# B&R Automation Studio project MySQLConnectorDemo
Automation Studio 4.12.6.106

## Configuration Config1

CPU X20CP3586, AutomationRuntime I4.93, Build 6.3.0, Vc 

### Task classes (Cpu.sw)
```
Cyclic#4:
  CmdGenerat <- MySQLInserter.CmdGenerator.prg
  Demo <- MySQLInserter.Demo.prg
  SqlWriter <- MySQLInserter.SqlWriter.prg
Binaries: udbdef, FWRules, TCData, sysconf, Role, User, iomap, ashwd, asfw, arconfig, ashwac
Libraries: AsBrStr, sys_lib, runtime, LxVar, asstring, astime, asieccon, BrRand, brsystem, standard
```

### Hardware
```
X20CP3586 : X20CP3586 v1.10.0.0
  Connector IF2:
    ActivateDevice = 1
    Mode = Manual
    InternetAddress = 192.168.0.200
    SubnetMask = 255.255.255.0
    ActivateSnmp = 2
  ConfigurationID = MySQLConnectorDemo_Config1
  RemanentGlobalPvSize = 80960
  FileDevice1
  FileDeviceName1 = USER
  FileDevicePath1 = USER_PATH
  ActivateOpcUa = 1
  OpcUaInformationModels_PV_Version = 1
```

### Config.mpdatabasecore - X20CP3586/mappServices/Config.mpdatabasecore
```
Element gDatabaseCore (Type=mpdatabasecore)
  mapp.Database.Core:
    Name = wn_9
    UserName = newuser
    Password = 123456
    PortNumber = 85
    DBQueries:
      [0]:
        Name = RdByTime
        Type = Custom
          Query = {&pv[gSqlStr]}
          Columns = SingleColumns
            [0]:
              Column = rdFloat1
              PV = ::SqlReader:RdBuffer.rdFloat1[]
            [1]:
              Column = rdFloat2
              PV = ::SqlReader:RdBuffer.rdFloat2[]
            [2]:
              Column = rdFloat3
              PV = ::SqlReader:RdBuffer.rdFloat3[]
      [1]:
        Name = RdByName
        Type = Custom
          Query = {&pv[gSqlStr]}
          Columns:
            PV = 
```

## Logical view

Binary libraries used (declarations not repeated): operator, runtime, astime, AsIecCon, AsBrStr, sys_lib, asstring, brsystem, standard, MpDatabase 5.24.3, BrRand

### Package Logical/Libraries - Global libraries

### GlobalMySQL.var
```iecst
VAR
	gMySQLInserter : MySQLInserter_typ;
END_VAR
VAR CONSTANT
	TASK_SIZE : USINT := 4;
	TASK_SIZE_MINUS_ONE : USINT := TASK_SIZE-1;
	INTERFACE_SIZE : USINT := 1;
	INTERFACE_SIZE_MINUS_ONE : USINT := INTERFACE_SIZE-1;
	CMD_STR_SIZE : UINT := 4000;
	SQL_NAME_STR_SIZE : USINT := 10;
	DATA_SIZE : USINT := 100;
	DATA_SIZE_MINUS_ONE : USINT := DATA_SIZE-1;
END_VAR
```

### GlobalMySQL.typ
```iecst
TYPE
	MySQLInserter_typ : 	STRUCT
		Command : MySQLInserterCommand_typ;
		Input : MySQLInserterInput_typ;
		Status : MySQLInserterStatus_typ;
		Config : MySQLInserterConfig_typ;
		ExternalCom : MySQLInserterExternalCom_typ;
		_Internal : MySQLInserterInternal_typ;
	END_STRUCT;
	MySQLInserterCommand_typ : 	STRUCT
		Enable : BOOL;
		Reset : BOOL;
	END_STRUCT;
	MySQLInserterInput_typ : 	STRUCT
		TaskTrig : ARRAY[0..TASK_SIZE_MINUS_ONE]OF BOOL;
	END_STRUCT;
	MySQLInserterStatus_typ : 	STRUCT
		BufferNum : ARRAY[0..INTERFACE_SIZE_MINUS_ONE]OF USINT;
		Connected : BOOL;
		Task : ARRAY[0..TASK_SIZE_MINUS_ONE]OF TaskStatus_typ;
	END_STRUCT;
	MySQLInserterConfig_typ : 	STRUCT
		TaskSetting : ARRAY[0..TASK_SIZE_MINUS_ONE]OF TaskSetting_typ;
		LostTimeMs : UDINT; (*Connect lost time*)
	END_STRUCT;
	MySQLInserterInternal_typ : 	STRUCT
		TaskCmdStr : ARRAY[0..TASK_SIZE_MINUS_ONE]OF STRING[CMD_STR_SIZE];
	END_STRUCT;
	MySQLInserterExternalCom_typ : 	STRUCT
		StrCmd : ARRAY[0..INTERFACE_SIZE_MINUS_ONE]OF STRING[CMD_STR_SIZE];
		Counter : ARRAY[0..INTERFACE_SIZE_MINUS_ONE]OF UDINT;
		HeartBeat : ARRAY[0..INTERFACE_SIZE_MINUS_ONE]OF UDINT;
	END_STRUCT;
	DataSetting_typ : 	STRUCT
		Name : STRING[SQL_NAME_STR_SIZE];
		Type : STRING[SQL_NAME_STR_SIZE];
		DataAddr : UDINT;
		DataSize : USINT; (*VARCHAR需要设置，DATETIME推荐设置*)
		Digital : USINT; (*仅FLOAT有效：
保留小数点位数*)
		ManualTime : BOOL; (*仅DATETIME有效:
0：自动生成TimeStamp
1：外部给出TimeStamp*)
		MissingCheck : BOOL; (*仅INT有效:(关联数据，外部请勿操作)
0：关闭
1：开启，默认自增1，用于检查是否漏写*)
		AutoIncrement : BOOL; (*mysql属性AUTO_INCREMENT*)
		NotNull : BOOL; (*mysql属性NOT NULL*)
		PrimaryKey : BOOL; (*mysql属性PRIMARY KEY*)
	END_STRUCT;
	MySQLInserterTask_typ : 	STRUCT
		Setting : TaskSetting_typ;
		Status : TaskStatus_typ;
	END_STRUCT;
	TaskStatus_typ : 	STRUCT
		Err : USINT;
		ErrMsg : STRING[64];
		CacheCount : USINT;
	END_STRUCT;
	TaskSetting_typ : 	STRUCT
		TrigMode : USINT; (*0：外部上升沿触发
1：按照采样时间自动触发*)
		IntervalTimeMs : UINT; (*采样间隔时间ms，最好不要<1000，最好是1000的整数倍*)
		DbName : STRING[SQL_NAME_STR_SIZE];
		TableName : STRING[SQL_NAME_STR_SIZE];
		CacheSize : USINT; (*缓存大小，设置合并插入*)
		WritePrimaryKey : USINT; (*是否写入主键*)
		DataSetting : ARRAY[0..DATA_SIZE_MINUS_ONE]OF DataSetting_typ;
	END_STRUCT;
END_TYPE
```

### Program Logical/MySQLInserter/CmdGenerator (ANSIC)

#### Variables.var - Local variables
```iecst
VAR
	InsCfg : REFERENCE TO MySQLInserterConfig_typ;
	InsSts : REFERENCE TO MySQLInserterStatus_typ;
	InsInter : REFERENCE TO MySQLInserterInternal_typ;
	InsInput : REFERENCE TO MySQLInserterInput_typ;
	InsCmd : REFERENCE TO MySQLInserterCommand_typ;
	u8idx : USINT;
	strBuffer : ARRAY[0..TASK_SIZE_MINUS_ONE] OF STRING[CMD_STR_SIZE];
	RTInfo_0 : RTInfo;
	accTimeUs : ARRAY[0..TASK_SIZE_MINUS_ONE] OF UDINT;
	firstScan : BOOL;
END_VAR
```

#### Main.c - Init, cyclic, exit code
```c
#include <bur/plctypes.h>
#include "SqlMaker.h"
#ifdef _DEFAULT_INCLUDES
	#include <AsDefault.h>
#endif

void _INIT ProgramInit(void)
{
	// Insert code here
	InsCfg = &gMySQLInserter.Config;
	InsSts = &gMySQLInserter.Status;
	InsInter = &gMySQLInserter._Internal;
	InsInput = &gMySQLInserter.Input;
	InsCmd = &gMySQLInserter.Command;
	firstScan = 1;
}

void _CYCLIC ProgramCyclic(void)
{
	// Insert code here
	if (0 == InsCmd->Enable) {
		return;
	}

	if (InsCmd->Reset) {
		firstScan = 1;
	}

	/* 获取线程信息 */
	RTInfo_0.enable = 1;
	RTInfo(&RTInfo_0);

	if (firstScan) {
		for (u8idx = 0; u8idx < TASK_SIZE ; u8idx++) {
			MakeCreateTableSql(strBuffer[u8idx], CMD_STR_SIZE, &InsCfg->TaskSetting[u8idx]);
			brsmemcpy((UDINT)InsInter->TaskCmdStr[u8idx], (UDINT)strBuffer[u8idx], CMD_STR_SIZE);
			InsSts->Task[u8idx].CacheCount = 0; // Cache清0
		}
		firstScan = 0;
		return;
	}

	for (u8idx = 0; u8idx < TASK_SIZE ; u8idx++) {
		// 定时触发模式
		if (1 == InsCfg->TaskSetting[u8idx].TrigMode) {
			if (InsCfg->TaskSetting[u8idx].IntervalTimeMs * 1000 > RTInfo_0.cycle_time && RTInfo_0.cycle_time != 0) {
				accTimeUs[u8idx] = accTimeUs[u8idx] + RTInfo_0.cycle_time;
				if (accTimeUs[u8idx] >= InsCfg->TaskSetting[u8idx].IntervalTimeMs * 1000){
					// 计时到，采集一次数据
					MakeInsertSql(strBuffer[u8idx], CMD_STR_SIZE, &InsCfg->TaskSetting[u8idx], &InsSts->Task[u8idx]);
					accTimeUs[u8idx] = 0;
				}
			} else {
				InsSts->Task[u8idx].Err = 1;
				strcpy(InsSts->Task[u8idx].ErrMsg, "Sampling interval is less than task cycle time.");
			}
		// 手动触发模式
		}else if (0 == InsCfg->TaskSetting[u8idx].TrigMode) {
			if (1 == InsInput->TaskTrig[u8idx]) {
				InsInput->TaskTrig[u8idx] = 0;
				MakeInsertSql(strBuffer[u8idx], CMD_STR_SIZE, &InsCfg->TaskSetting[u8idx], &InsSts->Task[u8idx]);
			}
		}
		// 到达cache_size大小，自动封包
		if (0 == InsSts->Task[u8idx].CacheCount) {
			// memset((UDINT)InsInter->TaskCmdStr[u8idx], 0, CMD_STR_SIZE);
			brsmemcpy((UDINT)InsInter->TaskCmdStr[u8idx], (UDINT)strBuffer[u8idx], CMD_STR_SIZE);
		}
	}
}

void _EXIT ProgramExit(void)
{
	// Insert code here

}
```

#### SqlMaker.h
```c
#ifndef SQLMAKER_H
#define SQLMAKER_H

#include <bur/plctypes.h>
#include <string.h>
#include <LxVar.h>

#ifdef _DEFAULT_INCLUDES
	#include <AsDefault.h>
#endif

void MakeInsertSql(STRING* sqlBuffer, UDINT bufferSize, TaskSetting_typ* taskSetting, TaskStatus_typ* taskStatus);
void MakeCreateTableSql(STRING* sqlBuffer, UDINT bufferSize, TaskSetting_typ* taskSetting);
UDINT CreateMySQLDateTimeStamp(STRING *pOutputString);

#endif // SQLMAKER_H
```

#### SqlMaker.c
```c
#include "SqlMaker.h"

void MakeInsertSql(STRING* sqlBuffer, UDINT bufferSize, TaskSetting_typ* taskSetting, TaskStatus_typ* taskStatus)
{
	// Calc data size
	if (0 == sizeof(taskSetting->DataSetting[0])) {
		return;
	}
	int dataSize = sizeof(taskSetting->DataSetting)/sizeof(taskSetting->DataSetting[0]);

	if (dataSize < 1) {
		return;
	}

	// Start building the SQL command
	if (0 == taskStatus->CacheCount) {
		memset((char*)sqlBuffer, 0, bufferSize);
		strcat((char*)sqlBuffer, "INSERT INTO ");
		strcat((char*)sqlBuffer, taskSetting->DbName);
		strcat((char*)sqlBuffer, ".");
		strcat((char*)sqlBuffer, taskSetting->TableName);
		strcat((char*)sqlBuffer, " (");

		// Add column names
		for (int i = 0; i < dataSize; ++i) {
			if (taskSetting->DataSetting[i].Name[0] == '\0') break;
			if (taskSetting->WritePrimaryKey == 0 && taskSetting->DataSetting[i].PrimaryKey == 1) {
				continue;
			}
			strcat((char*)sqlBuffer, taskSetting->DataSetting[i].Name);
			if (i < (dataSize - 1) && taskSetting->DataSetting[i+1].Name[0] != '\0') {
				strcat((char*)sqlBuffer, ",");
			}
		}
		strcat((char*)sqlBuffer, ") VALUES");
	}

	strcat((char*)sqlBuffer, "(");
	STRING tempStr[32];
	FB_Real2Str_typ FB_Real2Str_0;
	// Add value placeholders
	for (int i = 0; i < dataSize; ++i) {
		if (taskSetting->DataSetting[i].Name[0] == '\0') break;
		if (taskSetting->WritePrimaryKey == 0 && taskSetting->DataSetting[i].PrimaryKey == 1) {
			continue;
		}
		memset((char*)tempStr, 0, sizeof(tempStr));
		// Use '%s' for string, '%d' for int, etc. Here, just use '?' as placeholder
		if (strcmp(taskSetting->DataSetting[i].Type, "FLOAT") == 0) {
			// Type is FLOAT
			if (taskSetting->DataSetting[i].Digital != 0) {
				FB_Real2Str_0.digital = taskSetting->DataSetting[i].Digital;
				FB_Real2Str_0.rNum = *(REAL*)(taskSetting->DataSetting[i].DataAddr);
				FB_Real2Str(&FB_Real2Str_0);
				strcat((char*)tempStr, FB_Real2Str_0.strOut);
			}else {
				ftoa(*(REAL*)taskSetting->DataSetting[i].DataAddr, (UDINT)tempStr);
			}
			strcat((char*)sqlBuffer, (char*)tempStr);
		}
		else if (strcmp(taskSetting->DataSetting[i].Type, "INT") == 0) {
			// Type is INT
			if (1 == taskSetting->DataSetting[i].MissingCheck) {
				*(DINT*)taskSetting->DataSetting[i].DataAddr += 1;
			}
			itoa(*(DINT*)taskSetting->DataSetting[i].DataAddr, (UDINT)tempStr);
			strcat((char*)sqlBuffer, (char*)tempStr);
		}
		else if (strcmp(taskSetting->DataSetting[i].Type, "VARCHAR") == 0) {
			// Type is VARCHAR
			strcat((char*)sqlBuffer, (char*)taskSetting->DataSetting[i].DataAddr);
		}
		else if (strcmp(taskSetting->DataSetting[i].Type, "DATETIME") == 0) {
			// Type is DATETIME
			if (0 == taskSetting->DataSetting[i].ManualTime) {
				CreateMySQLDateTimeStamp(&tempStr);
				strcat((char*)sqlBuffer, (char*)tempStr);
			}else {
				strcat((char*)sqlBuffer, (char*)taskSetting->DataSetting[i].DataAddr);
			}
		}
		else {
			// Default case, treat as string
		}

		if (i < (dataSize - 1) && taskSetting->DataSetting[i+1].Name[0] != '\0') {
			strcat((char*)sqlBuffer, ",");
		}
	}
	strcat((char*)sqlBuffer, ")");
	if (taskStatus->CacheCount < (taskSetting->CacheSize - 1) && taskSetting->CacheSize != 0) {
		taskStatus->CacheCount = taskStatus->CacheCount + 1;
		strcat((char*)sqlBuffer, ",");
	} else {
		taskStatus->CacheCount = 0;
		strcat((char*)sqlBuffer, ";");
	}
}

void MakeCreateTableSql(STRING* sqlBuffer, UDINT bufferSize, TaskSetting_typ* taskSetting)
{
	if (0 == sizeof(taskSetting->DataSetting[0])) {
		return;
	}
	int dataSize = sizeof(taskSetting->DataSetting)/sizeof(taskSetting->DataSetting[0]);
	if (dataSize < 1) {
		return;
	}

	memset((char*)sqlBuffer, 0, bufferSize);
	strcat((char*)sqlBuffer, "CREATE TABLE IF NOT EXISTS ");
	strcat((char*)sqlBuffer, taskSetting->DbName);
	strcat((char*)sqlBuffer, ".");
	strcat((char*)sqlBuffer, taskSetting->TableName);
	strcat((char*)sqlBuffer, " (");

	for (int i = 0; i < dataSize; ++i) {
		if (taskSetting->DataSetting[i].Name[0] == '\0') {
			if (0 == i) {
				memset((char*)sqlBuffer, 0, bufferSize);
				return;
			}
			break;
		}
		strcat((char*)sqlBuffer, taskSetting->DataSetting[i].Name);
		strcat((char*)sqlBuffer, " ");
		strcat((char*)sqlBuffer, taskSetting->DataSetting[i].Type);

		// VARCHAR length
		if (strcmp(taskSetting->DataSetting[i].Type, "VARCHAR") == 0 && taskSetting->DataSetting[i].DataSize > 0) {
			char lenStr[8] = {0};
			strcat((char*)sqlBuffer, "(");
			itoa(taskSetting->DataSetting[i].DataSize, (UDINT)lenStr);
			strcat((char*)sqlBuffer, lenStr);
			strcat((char*)sqlBuffer, ")");
		}

		// Auto increment
		if (taskSetting->DataSetting[i].AutoIncrement) {
			strcat((char*)sqlBuffer, " AUTO_INCREMENT");
		}

		// NOT NULL
		if (taskSetting->DataSetting[i].NotNull) {
			strcat((char*)sqlBuffer, " NOT NULL");
		}

		// PRIMARY KEY
		if (taskSetting->DataSetting[i].PrimaryKey) {
			strcat((char*)sqlBuffer, " PRIMARY KEY");
		}

		if (i < (dataSize - 1) && taskSetting->DataSetting[i+1].Name[0] != '\0') {
			strcat((char*)sqlBuffer, ",");
		}
	}
	strcat((char*)sqlBuffer, ");");
}

UDINT CreateMySQLDateTimeStamp(STRING *pOutputString)
{
	STRING tempString[10];
	RTCtime_typ	RTC;

	/* Clear output string */
	memset(pOutputString, 0, sizeof(*pOutputString));
	/* Clear temp string */
	memset(&tempString, 0, sizeof(tempString));

	/* Get time */
	RTC_gettime(&RTC);

	/* copy in single quote */
	strcpy(pOutputString, "'");
	/* copy in year */
	itoa(RTC.year, (UDINT)tempString);
	strcat(pOutputString, tempString);
	/* add dash */
	strcat(pOutputString, "-");
	/* copy in month */
	itoa(RTC.month, (UDINT)tempString);
	strcat(pOutputString, tempString);
	/* add dash */
	strcat(pOutputString, "-");
	/* copy in day */
	itoa(RTC.day, (UDINT)tempString);
	strcat(pOutputString, tempString);

	/* add space */
	strcat(pOutputString, " ");

	/* copy in hour */
	itoa(RTC.hour, (UDINT)tempString);
	strcat(pOutputString, tempString);
	/* add colon */
	strcat(pOutputString, ":");
	/* copy in minutes */
	itoa(RTC.minute, (UDINT)tempString);
	strcat(pOutputString, tempString);
	/* add colon */
	strcat(pOutputString, ":");
	/* copy in seconds */
	itoa(RTC.second, (UDINT)tempString);
	strcat(pOutputString, tempString);
	/* copy in single quote */
	strcat(pOutputString, "'");

	return((UDINT)pOutputString);
}
```

### Program Logical/MySQLInserter/SqlWriter (ANSIC)

#### Variables.var - Local variables
```iecst
VAR
	InsInter : REFERENCE TO MySQLInserterInternal_typ;
	InsSts : REFERENCE TO MySQLInserterStatus_typ;
	InsExtCom : REFERENCE TO MySQLInserterExternalCom_typ;
	InsCmd : REFERENCE TO MySQLInserterCommand_typ;
	InsCfg : REFERENCE TO MySQLInserterConfig_typ;
	u8idx : USINT;
	step : USINT;
	oldCounter : UDINT;
	ton_0 : TON;
	ton_con : TON;
END_VAR
VAR CONSTANT
	INTERFACE_IDX : USINT := 0;
END_VAR
VAR
	oldTaskCmdStr : ARRAY[0..TASK_SIZE_MINUS_ONE] OF STRING[CMD_STR_SIZE];
	tempStr : {REDUND_UNREPLICABLE} STRING[10];
	oldHeartBeat : UDINT;
END_VAR
```

#### Main.c - Init, cyclic, exit code
```c
#include <bur/plctypes.h>
#include "deque.h"
#ifdef _DEFAULT_INCLUDES
#include <AsDefault.h>
#endif

_LOCAL Deque sqlDeque1;
_LOCAL DequeElement sqlElement1;

void _INIT ProgramInit(void)
{
	InsInter = &gMySQLInserter._Internal;
	InsSts = &gMySQLInserter.Status;
	InsExtCom = &gMySQLInserter.ExternalCom;
	InsCmd = &gMySQLInserter.Command;
	InsCfg = &gMySQLInserter.Config;
}

void _CYCLIC ProgramCyclic(void)
{
	if (0 == InsCmd->Enable) {
		return;
	}

	if (InsCmd->Reset) {
		step = 0;
	}

	switch(step) {
		case 0:
			// 初始化Deque
			initDeque(&sqlDeque1);

			memset(tempStr, 0, sizeof(tempStr));
			strcat(tempStr, "CREATE");
			step = 1;
			break;
		case 1:
			// 等待任务
			if(sqlDeque1.size > 0) {
				popDeque(&sqlDeque1, &sqlElement1);
				memcpy(InsExtCom->StrCmd[INTERFACE_IDX], sqlElement1.strBuffer, CMD_STR_SIZE);
				oldCounter = InsExtCom->Counter[INTERFACE_IDX];
				step = 2;
			}
			break;
		case 2:
			// 处理任务
			ton_0.IN = 1;
			ton_0.PT = 2000; // 2000ms
			// 超时未回复处理
			if (ton_0.Q) {
				ton_0.IN = 0;
				if (memcmp(InsExtCom->StrCmd[INTERFACE_IDX], tempStr, sizeof(tempStr)) != 0) {
					memcpy(sqlElement1.strBuffer, InsExtCom->StrCmd[INTERFACE_IDX], CMD_STR_SIZE);
					pushDeque(&sqlDeque1, &sqlElement1);
					step = 1;
				} else {
					step = 11;
				}

			}

			if (InsExtCom->Counter[INTERFACE_IDX] != oldCounter) {
				// 任务处理完成
				ton_0.IN = 0;
				step = 1;
			}
			break;
		case 3:
			// 任务完成，返回空闲
			step = 1;
			break;

		case 11:
			// 处理错误
			// 这里可以添加错误处理逻辑
			InsSts->Task[u8idx].Err = 1;
			strcpy(InsSts->Task[u8idx].ErrMsg, "Fault Error: Can not execute create cmd.");
			break;
		default:
			step = 0;
			break;
	}

	// 循环检查，如果数据变化，就把数据压入Deque
	for(u8idx = 0; u8idx < TASK_SIZE; u8idx++) {
		if(memcmp(oldTaskCmdStr[u8idx], InsInter->TaskCmdStr[u8idx], CMD_STR_SIZE) != 0) {
			memcpy(oldTaskCmdStr[u8idx], InsInter->TaskCmdStr[u8idx], CMD_STR_SIZE);

			memset(sqlElement1.strBuffer, 0, CMD_STR_SIZE);
			memcpy(sqlElement1.strBuffer, InsInter->TaskCmdStr[u8idx], CMD_STR_SIZE);

			pushDeque(&sqlDeque1, &sqlElement1);
		}
	}

	// connect status
	ton_con.IN = 1;
	ton_con.PT = InsCfg->LostTimeMs;

	if (ton_con.Q) {
		ton_con.IN = 0;
		if (InsExtCom->HeartBeat[INTERFACE_IDX] != oldHeartBeat) {
			InsSts->Connected = 1;
		}else {
			InsSts->Connected = 0;
		}
		oldHeartBeat = InsExtCom->HeartBeat[INTERFACE_IDX];
	}

	InsSts->BufferNum[INTERFACE_IDX] = sqlDeque1.size;
	// FB CALL
	TON(&ton_0);
	TON(&ton_con);

}

void _EXIT ProgramExit(void)
{

}
```

#### deque.h
```c
#ifndef __DEQUE_H__
#define __DEQUE_H__

#include <stdio.h>

#ifdef _DEFAULT_INCLUDES
	#include <AsDefault.h>
#endif

#define MAX_SIZE 100  // 定义队列的最大容量

typedef struct {
	STRING strBuffer[CMD_STR_SIZE+1];
} DequeElement;

typedef struct {
	DequeElement cmd_data[MAX_SIZE];  // 存储数据的数组
	int front;           // 指向队列的前端
	int rear;            // 指向队列的后端
	int size;  			 // 记录deue的大小
	int error_id;   	 // 报错标志位
} Deque;

// 初始化双端队列
void initDeque(Deque* deque);
// 判断队列是否为空
int isEmpty(Deque* deque);

// 判断队列是否满
int isFull(Deque* deque);

int getSize(Deque* deque);

// 从队列后端插入元素
void pushDeque(Deque* deque, DequeElement* data_ptr);

// 从队列前端删除元素
void popDeque(Deque* deque, DequeElement* data_ptr);

#endif
```

#### deque.c
```c
#include "deque.h"

// 初始化双端队列
void initDeque(Deque* deque) {
	deque->front = -1;  // 初始化front为-1，表示空
	deque->rear = -1;   // 初始化rear为-1，表示空
	deque->error_id = 0;
	deque->size = 0;
}

// 判断队列是否为空
int isEmpty(Deque* deque) {
	return (deque->size == 0);
}

// 判断队列是否满
int isFull(Deque* deque) {
	return ((deque->rear + 1) % MAX_SIZE == deque->front);
}

int getSize(Deque* deque) {
	return deque->size;
}

// 从队列后端插入元素
void pushDeque(Deque* deque, DequeElement* data_ptr) {
	if (isFull(deque)) {
		// printf("Deque is full!\n");
		return;
	}
	if (isEmpty(deque)) {
		deque->front = 0;  // 如果队列为空，设置front为0
	}
	deque->rear = (deque->rear + 1) % MAX_SIZE;  // 更新rear
	// brsmemset(deque->cmd_data, 0, sizeof(DequeElement));
	brsmemcpy(&deque->cmd_data[deque->rear], data_ptr, sizeof(DequeElement));  // 插入元素
	deque->size++;	// 增加大小
}

// 从队列前端删除元素
void popDeque(Deque* deque, DequeElement* data_ptr) {
	if (isEmpty(deque)) {
		//printf("Deque is empty!\n");
		// 若空，将传入的data_ptr清空
		brsmemset(data_ptr, 0, sizeof(DequeElement));
		return;  // 返回一个无效值
	}
	brsmemcpy(data_ptr, &deque->cmd_data[deque->front], sizeof(DequeElement));  // 获取front的值
	brsmemset(&deque->cmd_data[deque->front], 0, sizeof(DequeElement));
	if (deque->front == deque->rear) {  // 如果只有一个元素
		deque->front = deque->rear = -1;  // 重置队列
	} else {
		deque->front = (deque->front + 1) % MAX_SIZE;  // 更新front
	}

	deque->size--;
	return;  // 队列前端元素
}
```

### Program Logical/MySQLInserter/Demo (IEC)

#### Variables.var
```iecst
VAR
	IP1 : DINT;
	IP2 : DINT;
	FP2 : REAL;
END_VAR
(*Insert your comment here.*)
VAR
	ID : DINT;
	STATE : DINT;
	TimeStamp : STRING[32];
	CV : REAL;
	VPF : REAL;
	WT : REAL;
	F1 : REAL;
	F2 : REAL;
	F3 : REAL;
	F4 : REAL;
	F5 : REAL;
	F6 : REAL;
	F7 : REAL;
	F8 : REAL;
	F9 : REAL;
	F10 : REAL;
	F11 : REAL;
	F12 : REAL;
	F13 : REAL;
	F14 : REAL;
	F15 : REAL;
	FP : REAL;
	AP1 : REAL;
	BP1 : REAL;
	AP2 : REAL;
	ST1 : REAL;
	ST2 : REAL;
	ST3 : REAL;
	ST4 : REAL;
	ST5 : REAL;
	ST6 : REAL;
	ST7 : REAL;
	ST8 : REAL;
	ST9 : REAL;
	ST10 : REAL;
	ST11 : REAL;
	ST12 : REAL;
	ST13 : REAL;
	ST14 : REAL;
	ST15 : REAL;
	AIR : REAL;
	CP : REAL;
	CT : REAL;
	CRT : REAL;
	ES : REAL;
	FP1 : REAL;
	FT : REAL;
	FF : REAL;
	FC : DINT;
	HT1 : REAL;
	HT2 : REAL;
	HT3 : REAL;
	HT4 : REAL;
	HT5 : REAL;
	HT6 : REAL;
	HT7 : REAL;
	HT8 : REAL;
	HT9 : REAL;
	HT10 : REAL;
	HT11 : REAL;
	HT12 : REAL;
	HT13 : REAL;
	HT14 : REAL;
	HT15 : REAL;
	HT16 : REAL;
	HT17 : REAL;
	HT18 : REAL;
	HT19 : REAL;
	HT20 : REAL;
	MP : REAL;
	MT : REAL;
	MCT : REAL;
	MCP : REAL;
	EC : REAL;
	EST : REAL;
	ES1 : REAL;
	TC : REAL;
	TF : REAL;
	TW : REAL;
END_VAR
```

#### Main.st
```iecst
PROGRAM _INIT
	(* Insert code here *)
	gMySQLInserter.Command.Enable := 1;
	gMySQLInserter.Config.LostTimeMs := 2000;

	(***********************任务0**********************************)
	gMySQLInserter.Config.TaskSetting[0].DbName := 'wn_8';
	gMySQLInserter.Config.TaskSetting[0].TableName := 'ct_data';
	gMySQLInserter.Config.TaskSetting[0].TrigMode := 1; // 定时自动触发
	gMySQLInserter.Config.TaskSetting[0].IntervalTimeMs := 1000;
	gMySQLInserter.Config.TaskSetting[0].CacheSize := 2;

	gMySQLInserter.Config.TaskSetting[0].DataSetting[0].DataAddr := ADR(IP1);
	gMySQLInserter.Config.TaskSetting[0].DataSetting[0].Name := 'IP1';
	gMySQLInserter.Config.TaskSetting[0].DataSetting[0].Type := 'INT';
	gMySQLInserter.Config.TaskSetting[0].DataSetting[1].DataAddr := ADR(FP1);
	gMySQLInserter.Config.TaskSetting[0].DataSetting[1].Name := 'FP1';
	gMySQLInserter.Config.TaskSetting[0].DataSetting[1].Type := 'FLOAT';
	gMySQLInserter.Config.TaskSetting[0].DataSetting[1].Digital := 2;

	(***********************任务1**********************************)
	gMySQLInserter.Config.TaskSetting[1].DbName := 'wn_8';
	gMySQLInserter.Config.TaskSetting[1].TableName := 'ct_cip';
	gMySQLInserter.Config.TaskSetting[1].TrigMode := 0; // 外部上升沿触发
	gMySQLInserter.Config.TaskSetting[1].IntervalTimeMs := 0;
	gMySQLInserter.Config.TaskSetting[1].CacheSize := 1;

	gMySQLInserter.Config.TaskSetting[1].DataSetting[0].DataAddr := ADR(IP2);
	gMySQLInserter.Config.TaskSetting[1].DataSetting[0].Name := 'IP2';
	gMySQLInserter.Config.TaskSetting[1].DataSetting[0].Type := 'INT';
	gMySQLInserter.Config.TaskSetting[1].DataSetting[1].DataAddr := ADR(FP2);
	gMySQLInserter.Config.TaskSetting[1].DataSetting[1].Name := 'FP2';
	gMySQLInserter.Config.TaskSetting[1].DataSetting[1].Type := 'FLOAT';
	gMySQLInserter.Config.TaskSetting[1].DataSetting[1].Digital := 3;

	(***********************任务2**********************************)
	gMySQLInserter.Config.TaskSetting[2].DbName := 'wn_9';
	gMySQLInserter.Config.TaskSetting[2].TableName := 'ct_data';
	gMySQLInserter.Config.TaskSetting[2].TrigMode := 1; // 定时自动触发
	gMySQLInserter.Config.TaskSetting[2].IntervalTimeMs := 1000;
	gMySQLInserter.Config.TaskSetting[2].CacheSize := 2;

	gMySQLInserter.Config.TaskSetting[2].DataSetting[0].DataAddr := ADR(ID);
	gMySQLInserter.Config.TaskSetting[2].DataSetting[0].Name := 'ID';
	gMySQLInserter.Config.TaskSetting[2].DataSetting[0].Type := 'INT';
	gMySQLInserter.Config.TaskSetting[2].DataSetting[0].PrimaryKey := TRUE;
	gMySQLInserter.Config.TaskSetting[2].DataSetting[0].AutoIncrement := TRUE;
	gMySQLInserter.Config.TaskSetting[2].DataSetting[0].NotNull := TRUE;

	gMySQLInserter.Config.TaskSetting[2].DataSetting[1].DataAddr := ADR(STATE);
	gMySQLInserter.Config.TaskSetting[2].DataSetting[1].Name := 'STATE';
	gMySQLInserter.Config.TaskSetting[2].DataSetting[1].Type := 'INT';
	gMySQLInserter.Config.TaskSetting[2].DataSetting[1].MissingCheck := 1; // 调试用。用于设定检测漏写的标志位，自增1

	gMySQLInserter.Config.TaskSetting[2].DataSetting[2].DataAddr := ADR(TimeStamp);
	gMySQLInserter.Config.TaskSetting[2].DataSetting[2].Name := 'TimeStamp';
	gMySQLInserter.Config.TaskSetting[2].DataSetting[2].Type := 'DATETIME';
	gMySQLInserter.Config.TaskSetting[2].DataSetting[2].DataSize := SIZEOF(TimeStamp);
	gMySQLInserter.Config.TaskSetting[2].DataSetting[2].ManualTime := FALSE; // 自动模式，实际用不到本地TimeStamp

	// F1 ~ F15
	gMySQLInserter.Config.TaskSetting[2].DataSetting[3].DataAddr := ADR(F1);
	gMySQLInserter.Config.TaskSetting[2].DataSetting[3].Name := 'F1';
	gMySQLInserter.Config.TaskSetting[2].DataSetting[3].Type := 'FLOAT';
	gMySQLInserter.Config.TaskSetting[2].DataSetting[3].Digital := 3;

	gMySQLInserter.Config.TaskSetting[2].DataSetting[4].DataAddr := ADR(F2);
	gMySQLInserter.Config.TaskSetting[2].DataSetting[4].Name := 'F2';
	gMySQLInserter.Config.TaskSetting[2].DataSetting[4].Type := 'FLOAT';
	gMySQLInserter.Config.TaskSetting[2].DataSetting[4].Digital := 3;

	gMySQLInserter.Config.TaskSetting[2].DataSetting[5].DataAddr := ADR(F3);
	gMySQLInserter.Config.TaskSetting[2].DataSetting[5].Name := 'F3';
	gMySQLInserter.Config.TaskSetting[2].DataSetting[5].Type := 'FLOAT';
	gMySQLInserter.Config.TaskSetting[2].DataSetting[5].Digital := 3;

	gMySQLInserter.Config.TaskSetting[2].DataSetting[6].DataAddr := ADR(F4);
	gMySQLInserter.Config.TaskSetting[2].DataSetting[6].Name := 'F4';
	gMySQLInserter.Config.TaskSetting[2].DataSetting[6].Type := 'FLOAT';
	gMySQLInserter.Config.TaskSetting[2].DataSetting[6].Digital := 3;

	gMySQLInserter.Config.TaskSetting[2].DataSetting[7].DataAddr := ADR(F5);
	gMySQLInserter.Config.TaskSetting[2].DataSetting[7].Name := 'F5';
	gMySQLInserter.Config.TaskSetting[2].DataSetting[7].Type := 'FLOAT';
	gMySQLInserter.Config.TaskSetting[2].DataSetting[7].Digital := 3;

	gMySQLInserter.Config.TaskSetting[2].DataSetting[8].DataAddr := ADR(F6);
	gMySQLInserter.Config.TaskSetting[2].DataSetting[8].Name := 'F6';
	gMySQLInserter.Config.TaskSetting[2].DataSetting[8].Type := 'FLOAT';
	gMySQLInserter.Config.TaskSetting[2].DataSetting[8].Digital := 3;

	gMySQLInserter.Config.TaskSetting[2].DataSetting[9].DataAddr := ADR(F7);
	gMySQLInserter.Config.TaskSetting[2].DataSetting[9].Name := 'F7';
	gMySQLInserter.Config.TaskSetting[2].DataSetting[9].Type := 'FLOAT';
	gMySQLInserter.Config.TaskSetting[2].DataSetting[9].Digital := 3;

	gMySQLInserter.Config.TaskSetting[2].DataSetting[10].DataAddr := ADR(F8);
	gMySQLInserter.Config.TaskSetting[2].DataSetting[10].Name := 'F8';
	gMySQLInserter.Config.TaskSetting[2].DataSetting[10].Type := 'FLOAT';
	gMySQLInserter.Config.TaskSetting[2].DataSetting[10].Digital := 3;

	gMySQLInserter.Config.TaskSetting[2].DataSetting[11].DataAddr := ADR(F9);
	gMySQLInserter.Config.TaskSetting[2].DataSetting[11].Name := 'F9';
	gMySQLInserter.Config.TaskSetting[2].DataSetting[11].Type := 'FLOAT';
	gMySQLInserter.Config.TaskSetting[2].DataSetting[11].Digital := 3;

	gMySQLInserter.Config.TaskSetting[2].DataSetting[12].DataAddr := ADR(F10);
	gMySQLInserter.Config.TaskSetting[2].DataSetting[12].Name := 'F10';
	gMySQLInserter.Config.TaskSetting[2].DataSetting[12].Type := 'FLOAT';
	gMySQLInserter.Config.TaskSetting[2].DataSetting[12].Digital := 3;

	gMySQLInserter.Config.TaskSetting[2].DataSetting[13].DataAddr := ADR(F11);
	gMySQLInserter.Config.TaskSetting[2].DataSetting[13].Name := 'F11';
	gMySQLInserter.Config.TaskSetting[2].DataSetting[13].Type := 'FLOAT';
	gMySQLInserter.Config.TaskSetting[2].DataSetting[13].Digital := 3;

	gMySQLInserter.Config.TaskSetting[2].DataSetting[14].DataAddr := ADR(F12);
	gMySQLInserter.Config.TaskSetting[2].DataSetting[14].Name := 'F12';
	gMySQLInserter.Config.TaskSetting[2].DataSetting[14].Type := 'FLOAT';
	gMySQLInserter.Config.TaskSetting[2].DataSetting[14].Digital := 3;

	gMySQLInserter.Config.TaskSetting[2].DataSetting[15].DataAddr := ADR(F13);
	gMySQLInserter.Config.TaskSetting[2].DataSetting[15].Name := 'F13';
	gMySQLInserter.Config.TaskSetting[2].DataSetting[15].Type := 'FLOAT';
	gMySQLInserter.Config.TaskSetting[2].DataSetting[15].Digital := 3;

	gMySQLInserter.Config.TaskSetting[2].DataSetting[16].DataAddr := ADR(F14);
	gMySQLInserter.Config.TaskSetting[2].DataSetting[16].Name := 'F14';
	gMySQLInserter.Config.TaskSetting[2].DataSetting[16].Type := 'FLOAT';
	gMySQLInserter.Config.TaskSetting[2].DataSetting[16].Digital := 3;

	gMySQLInserter.Config.TaskSetting[2].DataSetting[17].DataAddr := ADR(F15);
	gMySQLInserter.Config.TaskSetting[2].DataSetting[17].Name := 'F15';
	gMySQLInserter.Config.TaskSetting[2].DataSetting[17].Type := 'FLOAT';
	gMySQLInserter.Config.TaskSetting[2].DataSetting[17].Digital := 3;

	// FP
	gMySQLInserter.Config.TaskSetting[2].DataSetting[18].DataAddr := ADR(FP);
	gMySQLInserter.Config.TaskSetting[2].DataSetting[18].Name := 'FP';
	gMySQLInserter.Config.TaskSetting[2].DataSetting[18].Type := 'FLOAT';
	gMySQLInserter.Config.TaskSetting[2].DataSetting[18].Digital := 3;

	// AP1, BP1, AP2
	gMySQLInserter.Config.TaskSetting[2].DataSetting[19].DataAddr := ADR(AP1);
	gMySQLInserter.Config.TaskSetting[2].DataSetting[19].Name := 'AP1';
	gMySQLInserter.Config.TaskSetting[2].DataSetting[19].Type := 'FLOAT';
	gMySQLInserter.Config.TaskSetting[2].DataSetting[19].Digital := 3;

	gMySQLInserter.Config.TaskSetting[2].DataSetting[20].DataAddr := ADR(BP1);
	gMySQLInserter.Config.TaskSetting[2].DataSetting[20].Name := 'BP1';
	gMySQLInserter.Config.TaskSetting[2].DataSetting[20].Type := 'FLOAT';
	gMySQLInserter.Config.TaskSetting[2].DataSetting[20].Digital := 3;

	gMySQLInserter.Config.TaskSetting[2].DataSetting[21].DataAddr := ADR(AP2);
	gMySQLInserter.Config.TaskSetting[2].DataSetting[21].Name := 'AP2';
	gMySQLInserter.Config.TaskSetting[2].DataSetting[21].Type := 'FLOAT';
	gMySQLInserter.Config.TaskSetting[2].DataSetting[21].Digital := 3;

	// ST1 ~ ST15
	gMySQLInserter.Config.TaskSetting[2].DataSetting[22].DataAddr := ADR(ST1);
	gMySQLInserter.Config.TaskSetting[2].DataSetting[22].Name := 'ST1';
	gMySQLInserter.Config.TaskSetting[2].DataSetting[22].Type := 'FLOAT';
	gMySQLInserter.Config.TaskSetting[2].DataSetting[22].Digital := 3;

	gMySQLInserter.Config.TaskSetting[2].DataSetting[23].DataAddr := ADR(ST2);
	gMySQLInserter.Config.TaskSetting[2].DataSetting[23].Name := 'ST2';
	gMySQLInserter.Config.TaskSetting[2].DataSetting[23].Type := 'FLOAT';
	gMySQLInserter.Config.TaskSetting[2].DataSetting[23].Digital := 3;

	gMySQLInserter.Config.TaskSetting[2].DataSetting[24].DataAddr := ADR(ST3);
	gMySQLInserter.Config.TaskSetting[2].DataSetting[24].Name := 'ST3';
	gMySQLInserter.Config.TaskSetting[2].DataSetting[24].Type := 'FLOAT';
	gMySQLInserter.Config.TaskSetting[2].DataSetting[24].Digital := 3;

	gMySQLInserter.Config.TaskSetting[2].DataSetting[25].DataAddr := ADR(ST4);
	gMySQLInserter.Config.TaskSetting[2].DataSetting[25].Name := 'ST4';
	gMySQLInserter.Config.TaskSetting[2].DataSetting[25].Type := 'FLOAT';
	gMySQLInserter.Config.TaskSetting[2].DataSetting[25].Digital := 3;

	gMySQLInserter.Config.TaskSetting[2].DataSetting[26].DataAddr := ADR(ST5);
	gMySQLInserter.Config.TaskSetting[2].DataSetting[26].Name := 'ST5';
	gMySQLInserter.Config.TaskSetting[2].DataSetting[26].Type := 'FLOAT';
	gMySQLInserter.Config.TaskSetting[2].DataSetting[26].Digital := 3;

	gMySQLInserter.Config.TaskSetting[2].DataSetting[27].DataAddr := ADR(ST6);
	gMySQLInserter.Config.TaskSetting[2].DataSetting[27].Name := 'ST6';
	gMySQLInserter.Config.TaskSetting[2].DataSetting[27].Type := 'FLOAT';
	gMySQLInserter.Config.TaskSetting[2].DataSetting[27].Digital := 3;

	gMySQLInserter.Config.TaskSetting[2].DataSetting[28].DataAddr := ADR(ST7);
	gMySQLInserter.Config.TaskSetting[2].DataSetting[28].Name := 'ST7';
	gMySQLInserter.Config.TaskSetting[2].DataSetting[28].Type := 'FLOAT';
	gMySQLInserter.Config.TaskSetting[2].DataSetting[28].Digital := 3;

	gMySQLInserter.Config.TaskSetting[2].DataSetting[29].DataAddr := ADR(ST8);
	gMySQLInserter.Config.TaskSetting[2].DataSetting[29].Name := 'ST8';
	gMySQLInserter.Config.TaskSetting[2].DataSetting[29].Type := 'FLOAT';
	gMySQLInserter.Config.TaskSetting[2].DataSetting[29].Digital := 3;

	gMySQLInserter.Config.TaskSetting[2].DataSetting[30].DataAddr := ADR(ST9);
	gMySQLInserter.Config.TaskSetting[2].DataSetting[30].Name := 'ST9';
	gMySQLInserter.Config.TaskSetting[2].DataSetting[30].Type := 'FLOAT';
	gMySQLInserter.Config.TaskSetting[2].DataSetting[30].Digital := 3;

	gMySQLInserter.Config.TaskSetting[2].DataSetting[31].DataAddr := ADR(ST10);
	gMySQLInserter.Config.TaskSetting[2].DataSetting[31].Name := 'ST10';
	gMySQLInserter.Config.TaskSetting[2].DataSetting[31].Type := 'FLOAT';
	gMySQLInserter.Config.TaskSetting[2].DataSetting[31].Digital := 3;

	gMySQLInserter.Config.TaskSetting[2].DataSetting[32].DataAddr := ADR(ST11);
	gMySQLInserter.Config.TaskSetting[2].DataSetting[32].Name := 'ST11';
	gMySQLInserter.Config.TaskSetting[2].DataSetting[32].Type := 'FLOAT';
	gMySQLInserter.Config.TaskSetting[2].DataSetting[32].Digital := 3;

	gMySQLInserter.Config.TaskSetting[2].DataSetting[33].DataAddr := ADR(ST12);
	gMySQLInserter.Config.TaskSetting[2].DataSetting[33].Name := 'ST12';
	gMySQLInserter.Config.TaskSetting[2].DataSetting[33].Type := 'FLOAT';
	gMySQLInserter.Config.TaskSetting[2].DataSetting[33].Digital := 3;

	gMySQLInserter.Config.TaskSetting[2].DataSetting[34].DataAddr := ADR(ST13);
	gMySQLInserter.Config.TaskSetting[2].DataSetting[34].Name := 'ST13';
	gMySQLInserter.Config.TaskSetting[2].DataSetting[34].Type := 'FLOAT';
	gMySQLInserter.Config.TaskSetting[2].DataSetting[34].Digital := 3;

	gMySQLInserter.Config.TaskSetting[2].DataSetting[35].DataAddr := ADR(ST14);
	gMySQLInserter.Config.TaskSetting[2].DataSetting[35].Name := 'ST14';
	gMySQLInserter.Config.TaskSetting[2].DataSetting[35].Type := 'FLOAT';
	gMySQLInserter.Config.TaskSetting[2].DataSetting[35].Digital := 3;

	gMySQLInserter.Config.TaskSetting[2].DataSetting[36].DataAddr := ADR(ST15);
	gMySQLInserter.Config.TaskSetting[2].DataSetting[36].Name := 'ST15';
	gMySQLInserter.Config.TaskSetting[2].DataSetting[36].Type := 'FLOAT';
	gMySQLInserter.Config.TaskSetting[2].DataSetting[36].Digital := 3;

	// AIR, CP, CT, CRT, ES, FP1, FT, FF
	gMySQLInserter.Config.TaskSetting[2].DataSetting[37].DataAddr := ADR(AIR);
	gMySQLInserter.Config.TaskSetting[2].DataSetting[37].Name := 'AIR';
	gMySQLInserter.Config.TaskSetting[2].DataSetting[37].Type := 'FLOAT';
	gMySQLInserter.Config.TaskSetting[2].DataSetting[37].Digital := 3;

	gMySQLInserter.Config.TaskSetting[2].DataSetting[38].DataAddr := ADR(CP);
	gMySQLInserter.Config.TaskSetting[2].DataSetting[38].Name := 'CP';
	gMySQLInserter.Config.TaskSetting[2].DataSetting[38].Type := 'FLOAT';
	gMySQLInserter.Config.TaskSetting[2].DataSetting[38].Digital := 3;

	gMySQLInserter.Config.TaskSetting[2].DataSetting[39].DataAddr := ADR(CT);
	gMySQLInserter.Config.TaskSetting[2].DataSetting[39].Name := 'CT';
	gMySQLInserter.Config.TaskSetting[2].DataSetting[39].Type := 'FLOAT';
	gMySQLInserter.Config.TaskSetting[2].DataSetting[39].Digital := 3;

	gMySQLInserter.Config.TaskSetting[2].DataSetting[40].DataAddr := ADR(CRT);
	gMySQLInserter.Config.TaskSetting[2].DataSetting[40].Name := 'CRT';
	gMySQLInserter.Config.TaskSetting[2].DataSetting[40].Type := 'FLOAT';
	gMySQLInserter.Config.TaskSetting[2].DataSetting[40].Digital := 3;

	gMySQLInserter.Config.TaskSetting[2].DataSetting[41].DataAddr := ADR(ES);
	gMySQLInserter.Config.TaskSetting[2].DataSetting[41].Name := 'ES';
	gMySQLInserter.Config.TaskSetting[2].DataSetting[41].Type := 'FLOAT';
	gMySQLInserter.Config.TaskSetting[2].DataSetting[41].Digital := 3;

	gMySQLInserter.Config.TaskSetting[2].DataSetting[42].DataAddr := ADR(FP1);
	gMySQLInserter.Config.TaskSetting[2].DataSetting[42].Name := 'FP1';
	gMySQLInserter.Config.TaskSetting[2].DataSetting[42].Type := 'FLOAT';
	gMySQLInserter.Config.TaskSetting[2].DataSetting[42].Digital := 3;

	gMySQLInserter.Config.TaskSetting[2].DataSetting[43].DataAddr := ADR(FT);
	gMySQLInserter.Config.TaskSetting[2].DataSetting[43].Name := 'FT';
	gMySQLInserter.Config.TaskSetting[2].DataSetting[43].Type := 'FLOAT';
	gMySQLInserter.Config.TaskSetting[2].DataSetting[43].Digital := 3;

	gMySQLInserter.Config.TaskSetting[2].DataSetting[44].DataAddr := ADR(FF);
	gMySQLInserter.Config.TaskSetting[2].DataSetting[44].Name := 'FF';
	gMySQLInserter.Config.TaskSetting[2].DataSetting[44].Type := 'FLOAT';
	gMySQLInserter.Config.TaskSetting[2].DataSetting[44].Digital := 3;

	// FC (DINT)
	gMySQLInserter.Config.TaskSetting[2].DataSetting[45].DataAddr := ADR(FC);
	gMySQLInserter.Config.TaskSetting[2].DataSetting[45].Name := 'FC';
	gMySQLInserter.Config.TaskSetting[2].DataSetting[45].Type := 'INT';

	// HT1 ~ HT20
	gMySQLInserter.Config.TaskSetting[2].DataSetting[46].DataAddr := ADR(HT1);
	gMySQLInserter.Config.TaskSetting[2].DataSetting[46].Name := 'HT1';
	gMySQLInserter.Config.TaskSetting[2].DataSetting[46].Type := 'FLOAT';
	gMySQLInserter.Config.TaskSetting[2].DataSetting[46].Digital := 3;

	gMySQLInserter.Config.TaskSetting[2].DataSetting[47].DataAddr := ADR(HT2);
	gMySQLInserter.Config.TaskSetting[2].DataSetting[47].Name := 'HT2';
	gMySQLInserter.Config.TaskSetting[2].DataSetting[47].Type := 'FLOAT';
	gMySQLInserter.Config.TaskSetting[2].DataSetting[47].Digital := 3;

	gMySQLInserter.Config.TaskSetting[2].DataSetting[48].DataAddr := ADR(HT3);
	gMySQLInserter.Config.TaskSetting[2].DataSetting[48].Name := 'HT3';
	gMySQLInserter.Config.TaskSetting[2].DataSetting[48].Type := 'FLOAT';
	gMySQLInserter.Config.TaskSetting[2].DataSetting[48].Digital := 3;

	gMySQLInserter.Config.TaskSetting[2].DataSetting[49].DataAddr := ADR(HT4);
	gMySQLInserter.Config.TaskSetting[2].DataSetting[49].Name := 'HT4';
	gMySQLInserter.Config.TaskSetting[2].DataSetting[49].Type := 'FLOAT';
	gMySQLInserter.Config.TaskSetting[2].DataSetting[49].Digital := 3;

	gMySQLInserter.Config.TaskSetting[2].DataSetting[50].DataAddr := ADR(HT5);
	gMySQLInserter.Config.TaskSetting[2].DataSetting[50].Name := 'HT5';
	gMySQLInserter.Config.TaskSetting[2].DataSetting[50].Type := 'FLOAT';
	gMySQLInserter.Config.TaskSetting[2].DataSetting[50].Digital := 3;

	gMySQLInserter.Config.TaskSetting[2].DataSetting[51].DataAddr := ADR(HT6);
	gMySQLInserter.Config.TaskSetting[2].DataSetting[51].Name := 'HT6';
	gMySQLInserter.Config.TaskSetting[2].DataSetting[51].Type := 'FLOAT';
	gMySQLInserter.Config.TaskSetting[2].DataSetting[51].Digital := 3;

	gMySQLInserter.Config.TaskSetting[2].DataSetting[52].DataAddr := ADR(HT7);
	gMySQLInserter.Config.TaskSetting[2].DataSetting[52].Name := 'HT7';
	gMySQLInserter.Config.TaskSetting[2].DataSetting[52].Type := 'FLOAT';
	gMySQLInserter.Config.TaskSetting[2].DataSetting[52].Digital := 3;

	gMySQLInserter.Config.TaskSetting[2].DataSetting[53].DataAddr := ADR(HT8);
	gMySQLInserter.Config.TaskSetting[2].DataSetting[53].Name := 'HT8';
	gMySQLInserter.Config.TaskSetting[2].DataSetting[53].Type := 'FLOAT';
	gMySQLInserter.Config.TaskSetting[2].DataSetting[53].Digital := 3;

	gMySQLInserter.Config.TaskSetting[2].DataSetting[54].DataAddr := ADR(HT9);
	gMySQLInserter.Config.TaskSetting[2].DataSetting[54].Name := 'HT9';
	gMySQLInserter.Config.TaskSetting[2].DataSetting[54].Type := 'FLOAT';
	gMySQLInserter.Config.TaskSetting[2].DataSetting[54].Digital := 3;

	gMySQLInserter.Config.TaskSetting[2].DataSetting[55].DataAddr := ADR(HT10);
	gMySQLInserter.Config.TaskSetting[2].DataSetting[55].Name := 'HT10';
	gMySQLInserter.Config.TaskSetting[2].DataSetting[55].Type := 'FLOAT';
	gMySQLInserter.Config.TaskSetting[2].DataSetting[55].Digital := 3;

	gMySQLInserter.Config.TaskSetting[2].DataSetting[56].DataAddr := ADR(HT11);
	gMySQLInserter.Config.TaskSetting[2].DataSetting[56].Name := 'HT11';
	gMySQLInserter.Config.TaskSetting[2].DataSetting[56].Type := 'FLOAT';
	gMySQLInserter.Config.TaskSetting[2].DataSetting[56].Digital := 3;

	gMySQLInserter.Config.TaskSetting[2].DataSetting[57].DataAddr := ADR(HT12);
	gMySQLInserter.Config.TaskSetting[2].DataSetting[57].Name := 'HT12';
	gMySQLInserter.Config.TaskSetting[2].DataSetting[57].Type := 'FLOAT';
	gMySQLInserter.Config.TaskSetting[2].DataSetting[57].Digital := 3;

	gMySQLInserter.Config.TaskSetting[2].DataSetting[58].DataAddr := ADR(HT13);
	gMySQLInserter.Config.TaskSetting[2].DataSetting[58].Name := 'HT13';
	gMySQLInserter.Config.TaskSetting[2].DataSetting[58].Type := 'FLOAT';
	gMySQLInserter.Config.TaskSetting[2].DataSetting[58].Digital := 3;

	gMySQLInserter.Config.TaskSetting[2].DataSetting[59].DataAddr := ADR(HT14);
	gMySQLInserter.Config.TaskSetting[2].DataSetting[59].Name := 'HT14';
	gMySQLInserter.Config.TaskSetting[2].DataSetting[59].Type := 'FLOAT';
	gMySQLInserter.Config.TaskSetting[2].DataSetting[59].Digital := 3;

	gMySQLInserter.Config.TaskSetting[2].DataSetting[60].DataAddr := ADR(HT15);
	gMySQLInserter.Config.TaskSetting[2].DataSetting[60].Name := 'HT15';
	gMySQLInserter.Config.TaskSetting[2].DataSetting[60].Type := 'FLOAT';
	gMySQLInserter.Config.TaskSetting[2].DataSetting[60].Digital := 3;

	gMySQLInserter.Config.TaskSetting[2].DataSetting[61].DataAddr := ADR(HT16);
	gMySQLInserter.Config.TaskSetting[2].DataSetting[61].Name := 'HT16';
	gMySQLInserter.Config.TaskSetting[2].DataSetting[61].Type := 'FLOAT';
	gMySQLInserter.Config.TaskSetting[2].DataSetting[61].Digital := 3;

	gMySQLInserter.Config.TaskSetting[2].DataSetting[62].DataAddr := ADR(HT17);
	gMySQLInserter.Config.TaskSetting[2].DataSetting[62].Name := 'HT17';
	gMySQLInserter.Config.TaskSetting[2].DataSetting[62].Type := 'FLOAT';
	gMySQLInserter.Config.TaskSetting[2].DataSetting[62].Digital := 3;

	gMySQLInserter.Config.TaskSetting[2].DataSetting[63].DataAddr := ADR(HT18);
	gMySQLInserter.Config.TaskSetting[2].DataSetting[63].Name := 'HT18';
	gMySQLInserter.Config.TaskSetting[2].DataSetting[63].Type := 'FLOAT';
	gMySQLInserter.Config.TaskSetting[2].DataSetting[63].Digital := 3;

	gMySQLInserter.Config.TaskSetting[2].DataSetting[64].DataAddr := ADR(HT19);
	gMySQLInserter.Config.TaskSetting[2].DataSetting[64].Name := 'HT19';
	gMySQLInserter.Config.TaskSetting[2].DataSetting[64].Type := 'FLOAT';
	gMySQLInserter.Config.TaskSetting[2].DataSetting[64].Digital := 3;

	gMySQLInserter.Config.TaskSetting[2].DataSetting[65].DataAddr := ADR(HT20);
	gMySQLInserter.Config.TaskSetting[2].DataSetting[65].Name := 'HT20';
	gMySQLInserter.Config.TaskSetting[2].DataSetting[65].Type := 'FLOAT';
	gMySQLInserter.Config.TaskSetting[2].DataSetting[65].Digital := 3;

	// MP, MT, MCT, MCP, EC, EST, ES1, TC, TF, TW
	gMySQLInserter.Config.TaskSetting[2].DataSetting[66].DataAddr := ADR(MP);
	gMySQLInserter.Config.TaskSetting[2].DataSetting[66].Name := 'MP';
	gMySQLInserter.Config.TaskSetting[2].DataSetting[66].Type := 'FLOAT';
	gMySQLInserter.Config.TaskSetting[2].DataSetting[66].Digital := 3;

	gMySQLInserter.Config.TaskSetting[2].DataSetting[67].DataAddr := ADR(MT);
	gMySQLInserter.Config.TaskSetting[2].DataSetting[67].Name := 'MT';
	gMySQLInserter.Config.TaskSetting[2].DataSetting[67].Type := 'FLOAT';
	gMySQLInserter.Config.TaskSetting[2].DataSetting[67].Digital := 3;

	gMySQLInserter.Config.TaskSetting[2].DataSetting[68].DataAddr := ADR(MCT);
	gMySQLInserter.Config.TaskSetting[2].DataSetting[68].Name := 'MCT';
	gMySQLInserter.Config.TaskSetting[2].DataSetting[68].Type := 'FLOAT';
	gMySQLInserter.Config.TaskSetting[2].DataSetting[68].Digital := 3;

	gMySQLInserter.Config.TaskSetting[2].DataSetting[69].DataAddr := ADR(MCP);
	gMySQLInserter.Config.TaskSetting[2].DataSetting[69].Name := 'MCP';
	gMySQLInserter.Config.TaskSetting[2].DataSetting[69].Type := 'FLOAT';
	gMySQLInserter.Config.TaskSetting[2].DataSetting[69].Digital := 3;

	gMySQLInserter.Config.TaskSetting[2].DataSetting[70].DataAddr := ADR(EC);
	gMySQLInserter.Config.TaskSetting[2].DataSetting[70].Name := 'EC';
	gMySQLInserter.Config.TaskSetting[2].DataSetting[70].Type := 'FLOAT';
	gMySQLInserter.Config.TaskSetting[2].DataSetting[70].Digital := 3;

	gMySQLInserter.Config.TaskSetting[2].DataSetting[71].DataAddr := ADR(EST);
	gMySQLInserter.Config.TaskSetting[2].DataSetting[71].Name := 'EST';
	gMySQLInserter.Config.TaskSetting[2].DataSetting[71].Type := 'FLOAT';
	gMySQLInserter.Config.TaskSetting[2].DataSetting[71].Digital := 3;

	gMySQLInserter.Config.TaskSetting[2].DataSetting[72].DataAddr := ADR(ES1);
	gMySQLInserter.Config.TaskSetting[2].DataSetting[72].Name := 'ES1';
	gMySQLInserter.Config.TaskSetting[2].DataSetting[72].Type := 'FLOAT';
	gMySQLInserter.Config.TaskSetting[2].DataSetting[72].Digital := 3;

	gMySQLInserter.Config.TaskSetting[2].DataSetting[73].DataAddr := ADR(TC);
	gMySQLInserter.Config.TaskSetting[2].DataSetting[73].Name := 'TC';
	gMySQLInserter.Config.TaskSetting[2].DataSetting[73].Type := 'FLOAT';
	gMySQLInserter.Config.TaskSetting[2].DataSetting[73].Digital := 3;

	gMySQLInserter.Config.TaskSetting[2].DataSetting[74].DataAddr := ADR(TF);
	gMySQLInserter.Config.TaskSetting[2].DataSetting[74].Name := 'TF';
	gMySQLInserter.Config.TaskSetting[2].DataSetting[74].Type := 'FLOAT';
	gMySQLInserter.Config.TaskSetting[2].DataSetting[74].Digital := 3;

	gMySQLInserter.Config.TaskSetting[2].DataSetting[75].DataAddr := ADR(TW);
	gMySQLInserter.Config.TaskSetting[2].DataSetting[75].Name := 'TW';
	gMySQLInserter.Config.TaskSetting[2].DataSetting[75].Type := 'FLOAT';
	gMySQLInserter.Config.TaskSetting[2].DataSetting[75].Digital := 3;

	gMySQLInserter.Config.TaskSetting[2].DataSetting[76].DataAddr := ADR(CV);
	gMySQLInserter.Config.TaskSetting[2].DataSetting[76].Name := 'CV';
	gMySQLInserter.Config.TaskSetting[2].DataSetting[76].Type := 'FLOAT';
	gMySQLInserter.Config.TaskSetting[2].DataSetting[76].Digital := 3;

	gMySQLInserter.Config.TaskSetting[2].DataSetting[77].DataAddr := ADR(VPF);
	gMySQLInserter.Config.TaskSetting[2].DataSetting[77].Name := 'VPF';
	gMySQLInserter.Config.TaskSetting[2].DataSetting[77].Type := 'FLOAT';
	gMySQLInserter.Config.TaskSetting[2].DataSetting[77].Digital := 3;
	// 添加 WT 点位
	gMySQLInserter.Config.TaskSetting[2].DataSetting[78].DataAddr := ADR(WT);
	gMySQLInserter.Config.TaskSetting[2].DataSetting[78].Name := 'WT';
	gMySQLInserter.Config.TaskSetting[2].DataSetting[78].Type := 'FLOAT';
	gMySQLInserter.Config.TaskSetting[2].DataSetting[78].Digital := 3;

END_PROGRAM

PROGRAM _CYCLIC
	(* Insert code here *)

	IP1 := RandINT();
	IP2 := RandINT();

	FP1 := RandRangeReal(0, 100);
	FP2 := RandRangeReal(0, 100);

	CV := RandRangeReal(0, 100);
	VPF := RandRangeReal(0, 100);
	WT := RandRangeReal(0, 100);

	F1 := RandRangeReal(0, 100);
	F2 := RandRangeReal(0, 100);
	F3 := RandRangeReal(0, 100);
	F4 := RandRangeReal(0, 100);
	F5 := RandRangeReal(0, 100);
	F6 := RandRangeReal(0, 100);
	F7 := RandRangeReal(0, 100);
	F8 := RandRangeReal(0, 100);
	F9 := RandRangeReal(0, 100);
	F10 := RandRangeReal(0, 100);
	F11 := RandRangeReal(0, 100);
	F12 := RandRangeReal(0, 100);
	F13 := RandRangeReal(0, 100);
	F14 := RandRangeReal(0, 100);
	F15 := RandRangeReal(0, 100);

	FP := RandRangeReal(0, 100);

	AP1 := RandRangeReal(0, 100);
	BP1 := RandRangeReal(0, 100);
	AP2 := RandRangeReal(0, 100);

	ST1 := RandRangeReal(0, 100);
	ST2 := RandRangeReal(0, 100);
	ST3 := RandRangeReal(0, 100);
	ST4 := RandRangeReal(0, 100);
	ST5 := RandRangeReal(0, 100);
	ST6 := RandRangeReal(0, 100);
	ST7 := RandRangeReal(0, 100);
	ST8 := RandRangeReal(0, 100);
	ST9 := RandRangeReal(0, 100);
	ST10 := RandRangeReal(0, 100);
	ST11 := RandRangeReal(0, 100);
	ST12 := RandRangeReal(0, 100);
	ST13 := RandRangeReal(0, 100);
	ST14 := RandRangeReal(0, 100);
	ST15 := RandRangeReal(0, 100);

	AIR := RandRangeReal(0, 100);
	CP := RandRangeReal(0, 100);
	CT := RandRangeReal(0, 100);
	CRT := RandRangeReal(0, 100);
	ES := RandRangeReal(0, 100);
	FT := RandRangeReal(0, 100);
	FF := RandRangeReal(0, 100);

	FC := RandINT();

	HT1 := RandRangeReal(0, 100);
	HT2 := RandRangeReal(0, 100);
	HT3 := RandRangeReal(0, 100);
	HT4 := RandRangeReal(0, 100);
	HT5 := RandRangeReal(0, 100);
	HT6 := RandRangeReal(0, 100);
	HT7 := RandRangeReal(0, 100);
	HT8 := RandRangeReal(0, 100);
	HT9 := RandRangeReal(0, 100);
	HT10 := RandRangeReal(0, 100);
	HT11 := RandRangeReal(0, 100);
	HT12 := RandRangeReal(0, 100);
	HT13 := RandRangeReal(0, 100);
	HT14 := RandRangeReal(0, 100);
	HT15 := RandRangeReal(0, 100);
	HT16 := RandRangeReal(0, 100);
	HT17 := RandRangeReal(0, 100);
	HT18 := RandRangeReal(0, 100);
	HT19 := RandRangeReal(0, 100);
	HT20 := RandRangeReal(0, 100);

	MP := RandRangeReal(0, 100);
	MT := RandRangeReal(0, 100);
	MCT := RandRangeReal(0, 100);
	MCP := RandRangeReal(0, 100);
	EC := RandRangeReal(0, 100);
	EST := RandRangeReal(0, 100);
	ES1 := RandRangeReal(0, 100);
	TC := RandRangeReal(0, 100);
	TF := RandRangeReal(0, 100);
	TW := RandRangeReal(0, 100);

	//gMySQLInserter.Task.Setting.DataSetting[]

END_PROGRAM

PROGRAM _EXIT
	(* Insert code here *)

END_PROGRAM
```

### Library Logical/MyLibraries/LxVar (ANSIC, version 1.00.4)
Depends on: AsBrStr, sys_lib

### Program Logical/mappDatabase/SqlReader (IEC)

#### Types.typ
```iecst
TYPE
	RdBuffer_typ : 	STRUCT
		rdFloat1 : ARRAY[0..MAX_FLOAT_NUM]OF REAL;
		rdFloat2 : ARRAY[0..MAX_FLOAT_NUM]OF REAL;
		rdFloat3 : ARRAY[0..MAX_FLOAT_NUM]OF REAL;
		rdFloat4 : ARRAY[0..MAX_FLOAT_NUM]OF REAL;
		rdFloat5 : ARRAY[0..MAX_FLOAT_NUM]OF REAL;
		rdFloat6 : ARRAY[0..MAX_FLOAT_NUM]OF REAL;
		rdFloat7 : ARRAY[0..MAX_FLOAT_NUM]OF REAL;
		rdInt1 : ARRAY[0..MAX_INT_NUM]OF DINT;
		rdInt2 : ARRAY[0..MAX_INT_NUM]OF DINT;
		rdInt3 : ARRAY[0..MAX_INT_NUM]OF DINT;
		rdInt4 : ARRAY[0..MAX_INT_NUM]OF DINT;
	END_STRUCT;
END_TYPE
```

#### Variables.var
```iecst
VAR CONSTANT
	MAX_INT_NUM : UINT := 37000;
	MAX_FLOAT_NUM : UINT := 37000;
END_VAR
VAR
	RdBuffer : RdBuffer_typ;
END_VAR
```

#### Main.st
```iecst
PROGRAM _INIT
	(* Insert code here *)

END_PROGRAM

PROGRAM _CYCLIC
	(* Insert code here *)
	Database;
	RdBuffer;
	gSqlStr;
END_PROGRAM

PROGRAM _EXIT
	(* Insert code here *)

END_PROGRAM
```

### Program Logical/mappDatabase/mappDB (IEC)

#### LocalVariables.var
```iecst
(*------------------------------------------------------------------------------------------------------------------------------------------------------------------------------------------------------------------------*)
(*SQL function calls*)
VAR
	MpDatabaseCore_0 : MpDatabaseCore; (*mappDatabase main function block*)
	MpDatabaseQuery_0 : MpDatabaseQuery; (*mappDatabase query*)
END_VAR
(*------------------------------------------------------------------------------------------------------------------------------------------------------------------------------------------------------------------------*)
VAR
	MpCfgRW_01 : MpCfgRW; (*Functionblock for mapp configuration read/write*)
	IcmpPing_0 : IcmpPing; (*Ping network share*)
	PingTimer : TON_10ms;
	PING_TIMEOUT : UINT := 200; (*Timeout for ping response*)
END_VAR
(*------------------------------------------------------------------------------------------------------------------------------------------------------------------------------------------------------------------------*)
(*Local variables*)
VAR
	SqlTimeout : TON_10ms; (*Timeout for SQL commands*)
	dbState : dbState_Enum; (*State machine*)
END_VAR
(*------------------------------------------------------------------------------------------------------------------------------------------------------------------------------------------------------------------------*)
(*Configuration for database managment*)
VAR CONSTANT
	TIMEOUT : UINT := 500; (*Timeout for SQL connection and query, default is 1000=>10s*)
END_VAR
(*------------------------------------------------------------------------------------------------------------------------------------------------------------------------------------------------------------------------*)
(*Local constants*)
VAR CONSTANT
	ERR_SQL_TIMEOUT_CONNECT : UINT := 10000; (*Timeout error for SQL connection*)
	ERR_SQL_TIMEOUT_QUERY : UINT := 10001; (*Timeout error for SQL query*)
	ERR_SQL_NOT_CONNECTED : UINT := 10010; (*Can not execute when not connected*)
END_VAR
```

#### Main.st
```iecst
PROGRAM _INIT
	// --------------------------------------------------------------------------------------------------------------------
	// Preset function blocks
	MpDatabaseCore_0.MpLink := ADR(gDatabaseCore);
	MpDatabaseQuery_0.MpLink := ADR(gDatabaseCore);

	SqlTimeout.PT := TIMEOUT;

	REPEAT
		MpCfgRW_01.Enable 		:= TRUE;
		MpCfgRW_01.MpLink 		:= gDatabaseCore;
		MpCfgRW_01.ReadWrite 	:= MpCfgRead;
		MpCfgRW_01.ParaName 	:= 'IPAddress';
		MpCfgRW_01.GroupArray	:= 0;
		MpCfgRW_01();
		UNTIL MpCfgRW_01.CommandDone
	END_REPEAT;

END_PROGRAM

PROGRAM _CYCLIC
	gSqlStr;
		// Trigger ping request
	PingTimer.IN := TRUE;
	PingTimer.PT := PING_TIMEOUT;
	PingTimer();
	// Try to ping network share if not connected
	IF(MpCfgRW_01.Value <> '' AND PingTimer.Q) THEN
		IcmpPing_0(enable := 1, pHost := ADR(MpCfgRW_01.Value), timeout := PING_TIMEOUT);
		// Ping was OK
		IF(IcmpPing_0.status = ERR_OK) THEN
			PingTimer(IN := FALSE);
			Database.PAR.CanPing := TRUE;
			// Disconnect from share when ping failed
		ELSIF(IcmpPing_0.status <> ERR_FUB_BUSY) THEN
			PingTimer(IN := FALSE);
			Database.PAR.CanPing := FALSE;
			IF(Database.PAR.IsConnected) THEN
				Database.CMD.Disconnect := TRUE;
			END_IF
		END_IF
	ELSIF(PingTimer.Q) THEN
		PingTimer(IN := FALSE);
	END_IF

	// --------------------------------------------------------------------------------------------------------------------
	// Database state machine
	// --------------------------------------------------------------------------------------------------------------------
	CASE dbState OF
		// --------------------------------------------------------------------------------------------------------------------
		// Wait state
		dbSTATE_WAIT:
			// --------------------------------------------------------------------------------------------------------------------
			// Connect to database
			IF Database.CMD.Connect THEN
				dbState := dbSTATE_CONNECT;
			END_IF

			// Disconnect from database
			IF Database.CMD.Disconnect THEN
				dbState := dbSTATE_DISCONNECT;
			END_IF

			// Execute SQL command
			IF Database.CMD.Execute THEN
				dbState := dbSTATE_QUERY;
			END_IF

			// Get next entry
			IF Database.CMD.NextRow THEN
				dbState := dbSTATE_NEXT;
			END_IF

			// --------------------------------------------------------------------------------------------------------------------
			// Reset error information and timeout timer
			IF Database.CMD.Connect OR Database.CMD.Disconnect OR Database.CMD.Execute OR Database.CMD.NextRow THEN
				Database.ERR.No := 0;
				brsmemset(ADR(Database.ERR.Text), 0, SIZEOF(Database.ERR.Text));

				MpDatabaseCore_0.Enable := TRUE;
				MpDatabaseQuery_0.Enable := TRUE;
				MpDatabaseQuery_0.ErrorReset := TRUE;
				MpDatabaseCore_0.ErrorReset := TRUE;
				MpDatabaseQuery_0();
				MpDatabaseCore_0();

				SqlTimeout.IN := 0;
				SqlTimeout();
			END_IF

		// --------------------------------------------------------------------------------------------------------------------
		// Connect state
		dbSTATE_CONNECT:
			SqlTimeout.IN := 1;
			SqlTimeout();

			IF MpDatabaseCore_0.CommandDone OR MpDatabaseCore_0.Error THEN
				IF MpDatabaseCore_0.Error THEN
					Database.ERR.No := MpDatabaseCore_0.StatusID;
					dbState := dbSTATE_ERROR;
				ELSE
					Database.CMD.Connect := FALSE;
					dbState := dbSTATE_WAIT;
				END_IF
			ELSIF SqlTimeout.Q THEN
				Database.ERR.No := ERR_SQL_TIMEOUT_CONNECT;
				MpDatabaseCore_0.Enable := FALSE;
				dbState := dbSTATE_ERROR;
			END_IF

		// --------------------------------------------------------------------------------------------------------------------
		// Disconnect state
		dbSTATE_DISCONNECT:
			SqlTimeout.IN := 1;
			SqlTimeout();

			IF MpDatabaseCore_0.CommandDone OR MpDatabaseCore_0.Error THEN

				IF MpDatabaseCore_0.Error THEN
					Database.ERR.No := MpDatabaseCore_0.StatusID;
					dbState := dbSTATE_ERROR;
				ELSE
					Database.CMD.Disconnect := FALSE;
					dbState := dbSTATE_WAIT;
				END_IF
			ELSIF SqlTimeout.Q THEN
				Database.ERR.No := ERR_SQL_TIMEOUT_CONNECT;
				MpDatabaseCore_0.Enable := FALSE;
				dbState := dbSTATE_ERROR;
			END_IF

		// --------------------------------------------------------------------------------------------------------------------
		// Query state
		dbSTATE_QUERY:
			SqlTimeout.IN := 1;
			SqlTimeout();

			IF MpDatabaseQuery_0.CommandDone OR MpDatabaseQuery_0.Error THEN
				Database.CMD.Execute := FALSE;

				IF MpDatabaseQuery_0.Error THEN
					Database.ERR.No := MpDatabaseQuery_0.StatusID;
					dbState := dbSTATE_ERROR;
				ELSE
					dbState := dbSTATE_WAIT;
				END_IF
			ELSIF NOT Database.PAR.IsConnected THEN
				Database.ERR.No := ERR_SQL_NOT_CONNECTED;
				dbState := dbSTATE_ERROR;
			ELSIF SqlTimeout.Q THEN
				Database.ERR.No := ERR_SQL_TIMEOUT_QUERY;
				MpDatabaseQuery_0.Enable := FALSE;
				dbState := dbSTATE_ERROR;
			END_IF

		// --------------------------------------------------------------------------------------------------------------------
		// Read next row
		dbSTATE_NEXT:
			SqlTimeout.IN := 1;
			SqlTimeout();

			IF MpDatabaseQuery_0.CommandDone OR MpDatabaseQuery_0.Error THEN
				Database.CMD.NextRow := FALSE;

				IF MpDatabaseQuery_0.Error THEN
					Database.ERR.No := MpDatabaseQuery_0.StatusID;
					dbState := dbSTATE_ERROR;
				ELSE
					dbState := dbSTATE_WAIT;
				END_IF
			ELSIF SqlTimeout.Q THEN
				Database.ERR.No := ERR_SQL_TIMEOUT_QUERY;
				MpDatabaseQuery_0.Enable := FALSE;
				dbState := dbSTATE_ERROR;
			END_IF

		// --------------------------------------------------------------------------------------------------------------------
		// Error state
		dbSTATE_ERROR:
			Database.CMD.Connect := FALSE;
			Database.CMD.Disconnect := FALSE;
			Database.CMD.Execute := FALSE;
			Database.CMD.NextRow := FALSE;

			IF Database.ERR.No = mpDATABASE_ERR_SQL_SERVER THEN
				Database.ERR.Text := 'Error response from SQL server. Check SQL syntax!';
			ELSIF Database.ERR.No = mpCOM_ERR_ACTIVATION THEN
				Database.ERR.Text := 'Could not create component query. Try to reboot PLC and script!';
			ELSIF Database.ERR.No = mpDATABASE_ERR_QUERY_RESULT THEN
				Database.ERR.Text := 'Check the query to determine if correct table and column names were used.';
			ELSIF Database.ERR.No = mpDATABASE_INF_NO_DATA THEN
				Database.ERR.Text := 'No more data available.';
			ELSIF Database.ERR.No = mpDATABASE_ERR_HTTP_SERVER AND NOT Database.PAR.IsConnected THEN
				Database.ERR.Text := 'Not connected to database. Try to reboot PLC and script!';
			ELSIF Database.ERR.No = ERR_SQL_TIMEOUT_CONNECT THEN
				Database.ERR.Text := 'SQL timeout during connection. Make sure script and server is running.';
			ELSIF Database.ERR.No = ERR_SQL_TIMEOUT_QUERY THEN
				Database.ERR.Text := 'SQL timeout during query.';
			ELSIF Database.ERR.No = ERR_SQL_NOT_CONNECTED THEN
				Database.ERR.Text := 'Not connected to database. Call command connect first';
			ELSE
				Database.ERR.Text := 'Generic SQL error.';
			END_IF

			dbState := dbSTATE_WAIT;
	END_CASE;

	// --------------------------------------------------------------------------------------------------------------------
	// Function block calls
	IF NOT MpDatabaseQuery_0.ErrorReset THEN
		MpDatabaseQuery_0.Execute := Database.CMD.Execute;
		MpDatabaseQuery_0.Next := Database.CMD.NextRow;
		MpDatabaseQuery_0.Name := ADR(Database.PAR.QueryName);
	END_IF
	MpDatabaseQuery_0();

	IF NOT MpDatabaseCore_0.ErrorReset THEN
		MpDatabaseCore_0.Connect := Database.CMD.Connect;
		MpDatabaseCore_0.Disconnect := Database.CMD.Disconnect;
	END_IF
	MpDatabaseCore_0();

	// Transfer function block data to global structure
	Database.PAR.IsConnected := MpDatabaseCore_0.Connected;
	Database.PAR.RowsTotal := MpDatabaseQuery_0.Info.Rows.Total;
	Database.PAR.RowsRead := MpDatabaseQuery_0.Info.Rows.Read;
	Database.PAR.RowsRemaining := MpDatabaseQuery_0.Info.Rows.Remaining;

	// Clear error reset command
	MpDatabaseQuery_0.ErrorReset := FALSE;
	MpDatabaseCore_0.ErrorReset := FALSE;

END_PROGRAM

PROGRAM _EXIT
	// --------------------------------------------------------------------------------------------------------------------
	// Exit function blocks
	MpDatabaseCore_0.Enable := FALSE;
	MpDatabaseCore_0();

	MpDatabaseQuery_0.Enable := FALSE;
	MpDatabaseQuery_0();

END_PROGRAM
```

### Program Logical/mappDatabase/RecipeSample (IEC)

#### Main.st
```iecst
PROGRAM _INIT
END_PROGRAM

PROGRAM _CYCLIC
	// Generate a list with all recipe names
	IF EDGEPOS(Database.PAR.IsConnected) THEN
		Recipe.CMD.List := TRUE;
	END_IF
	IF EDGEPOS(Recipe.CMD.List) THEN
		Database.PAR.QueryName := 'RecipeList';
		Database.CMD.Execute := TRUE;
		idx := 0;
		brsmemset(ADR(Recipe.PAR.RecipeNames), 0, SIZEOF(Recipe.PAR.RecipeNames));
	END_IF
	// Translate recipe names to mappView data providers
	IF Recipe.CMD.List AND (EDGENEG(Database.CMD.Execute) OR EDGENEG(Database.CMD.NextRow)) THEN
		brsstrcpy(ADR(Recipe.PAR.RecipeNames[idx]), ADR('{"value":"'));
		brsstrcat(ADR(Recipe.PAR.RecipeNames[idx]), ADR(Recipe.DATA.product_name));
		brsstrcat(ADR(Recipe.PAR.RecipeNames[idx]), ADR('","text":"'));
		brsstrcat(ADR(Recipe.PAR.RecipeNames[idx]), ADR(Recipe.DATA.product_name));
		brsstrcat(ADR(Recipe.PAR.RecipeNames[idx]), ADR('"}'));

		// Read next entry as long as we have entries and space
		IF Database.PAR.RowsRemaining > 0 AND idx < SIZEOF(Recipe.PAR.RecipeNames)/SIZEOF(Recipe.PAR.RecipeNames[idx]) THEN
			idx := idx + 1;
			Database.CMD.NextRow := TRUE;
		ELSE
			Recipe.CMD.List := FALSE;
		END_IF
	END_IF

	// Load recipe
	IF Recipe.CMD.Load THEN
		// Reset command
		IF EDGENEG(Database.CMD.Execute) THEN
			Recipe.CMD.Load := FALSE;
		// Trigger database command
		ELSE
			Database.PAR.QueryName := 'RecipeLoad';
			Database.CMD.Execute := TRUE;
		END_IF
	END_IF

	// Save recipe
	IF Recipe.CMD.Save OR Recipe.CMD.Rename THEN
		// Reset command
		IF EDGENEG(Database.CMD.Execute) THEN
			Recipe.CMD.Save := FALSE;
			IF Recipe.CMD.Rename THEN
				Recipe.CMD.Rename := FALSE;
				Recipe.CMD.List := TRUE;
			END_IF
		// Trigger database command
		ELSE
			Database.PAR.QueryName := 'RecipeSave';
			Database.CMD.Execute := TRUE;
		END_IF
	END_IF

	// New recipe
	IF Recipe.CMD.New THEN
		// Reset command
		IF EDGENEG(Database.CMD.Execute) THEN
			Recipe.CMD.New := FALSE;
			Recipe.CMD.List := TRUE;
		// Trigger database command
		ELSE
			Database.PAR.QueryName := 'RecipeNew';
			Database.CMD.Execute := TRUE;
		END_IF
	END_IF

	// Delete recipe
	IF Recipe.CMD.Delete THEN
		// Reset command
		IF EDGENEG(Database.CMD.Execute) THEN
			Recipe.CMD.Delete := FALSE;
			Recipe.CMD.List := TRUE;
		// Trigger database command
		ELSE
			Database.PAR.QueryName := 'RecipeDelete';
			Database.CMD.Execute := TRUE;
		END_IF
	END_IF

END_PROGRAM
```

### dbVariables.var
```iecst
VAR
	Database : dbMAIN; (*Database main structure*)
	Recipe : recMAIN; (*Recipe sample structure*)
	gSqlStr : STRING[500];
END_VAR
```

### changelog.txt
```
Version 1.2 (10.02.2023)
- PythonScript: Support for MS SQL data type decimal

Version 1.1 (05.01.2022)
- Added script server ping
- PLC: Update to runtime E4.90 and mapp 5.16
- PythonScript: Added PLC raw data to debug output

Version 1.0 (18.08.2021)
- PythonScript: Added more and detailed debug output
- PythonScript: Added more and detailed error messages
- PythonScript: Print all SQL queries and server response details
- PythonScript: Trim data type string when reading from database
- PythonScript: Change MsSQL database provider to 'ODBC Driver 17 for SQL Server' to support Linux systems
- PythonScript: Removed dependency from MySql driver for data conversion. Removed dependecy from MySql driver for data conversion. It is no longer required to install MySQL driver when using MsSQL.
```

Listed in the project but not available here: Logical/Global.typ, Logical/Global.var, Logical/MySQLInserter/CmdGenerator/Types.typ, Logical/MySQLInserter/SqlWriter/Types.typ, Logical/MyLibraries/LxVar/Types.typ, Logical/MyLibraries/LxVar/Constants.var, Logical/MyLibraries/LxVar/LxVar.fun, Logical/MyLibraries/LxVar/FB_GetPvInfo.c, Logical/MyLibraries/LxVar/GetPvOutside.c, Logical/MyLibraries/LxVar/DataJoint.c, Logical/MyLibraries/LxVar/DataSeparate.c, Logical/MyLibraries/LxVar/JudgeSrcPvInfoNum.c, Logical/MyLibraries/LxVar/FB_GetModuleName.c, Logical/MyLibraries/LxVar/FB_GetLocalPvAddr.c, Logical/MyLibraries/LxVar/FB_GetPvAddrStr.c, Logical/MyLibraries/LxVar/FB_GetStruPvMemName.c, Logical/MyLibraries/LxVar/FB_ShowPvAddrData.c, Logical/MyLibraries/LxVar/FB_ShowAddrData.c, Logical/MyLibraries/LxVar/FB_ShowLocalPvAddrData.c, Logical/MyLibraries/LxVar/Strcats.c, Logical/MyLibraries/LxVar/Strcpys.c, Logical/MyLibraries/LxVar/Strlens.c, Logical/MyLibraries/LxVar/FB_Udint2Str.c, Logical/MyLibraries/LxVar/VarWarnLogWrite.c, Logical/MyLibraries/LxVar/VarServLogWrite.c, Logical/MyLibraries/LxVar/FB_GetPvEntireName.c, Logical/MyLibraries/LxVar/ReturnPvAddr.c, Logical/MyLibraries/LxVar/FB_ContinualStrcat.c, Logical/mappDatabase/dbTypes.typ
